Staubli VAL3: product.dtx

mdesc mNomSpeed
public num nPeak
public frame fFrmMaster = {fatherId=world[0]}
public pointRx pDemo = {fatherId=fFrmMaster[0]}
public mdesc mNormal = {accel=20, decel=20, tmax=100, leave=1, reach=1, blend=cartesian}
public mdesc mJoint
public string sFrameName
public string sToolName
public string sPtParameter
public string sJtParameter
public tool tTool = {fatherId=flange[0], ioLink=valve1}
